PROGRAM main
  VAR
    DI_SensorPresence AT %QX0.3 : BOOL;
    DI_SensorHeight AT %QX0.4 : BOOL;
    DO_ConveyorMain AT %QX0.0 : BOOL;
    DO_ConveyorDivert AT %QX0.1 : BOOL;
    DO_Pusher AT %QX0.2 : BOOL;
    TimerPusher : TP;
    TP0 : TP;
  END_VAR

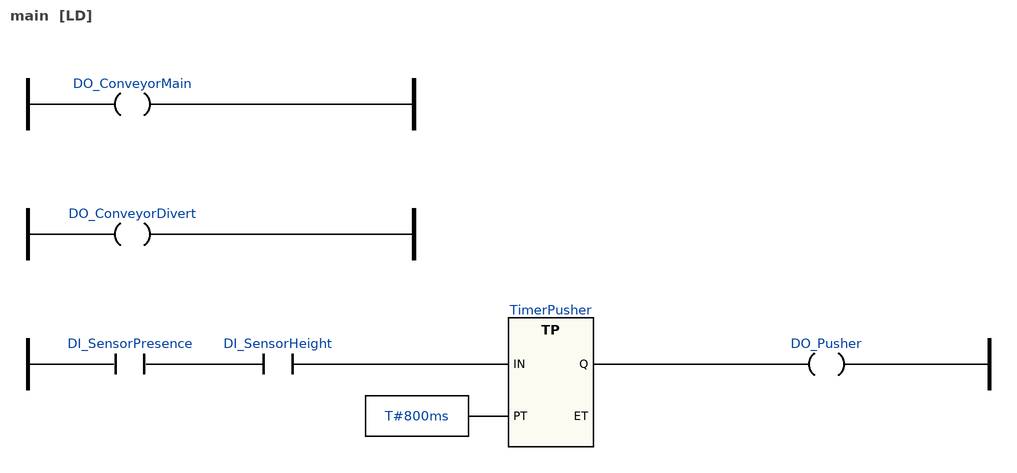
(* LD diagram, written out as Structured Text *)
DO_ConveyorMain := TRUE;
DO_ConveyorDivert := TRUE;
TimerPusher(IN := DI_SensorPresence AND DI_SensorHeight, PT := T#800ms);
DO_Pusher := TimerPusher.Q;
END_PROGRAM
